// TIA Portal project "traffic_light" (V17)

(* hardware
DEVICE "S7-1200 station_1"  S7-1200 Station
   slot 0: "Rack_0"  S7-1200 Rack  Rack  V1.0
   slot 1: "PLC_1"  CPU 1212C DC/DC/DC  6ES7 212-1AE40-0XB0  V4.1
DEVICE "HMI_1"  TP700 Comfort
   slot 0: "HMI_1"  TP700 Comfort  6AV2 124-0GC01-0AX0  17.0.0.0
   slot 1: "HMI_RT_1"  TP700 Comfort  6AV2 124-0GC01-0AX0  17.0.0.0
   slot 5: "HMI_1.IE_CP_1"  PROFINET Interface  17.0.0.0
      slot 1: "PROFINET Interface_1"  PROFINET Interface
         slot 1: "Port_1"  Port
         slot 2: "Port_2"  Port
   slot 7: "HMI_1.MPI/DP_CP_1"  MPI/DP Interface  17.0.0.0
*)

// ===== PLC "PLC_1"  CPU 1212C DC/DC/DC =====

VAR_GLOBAL   // PLC tag table "Tag table_1"
   "START" AT %M0.0 : Bool;
   "STOP" AT %M0.1 : Bool;
   "STARTED" AT %M0.2 : Bool;
   "STEP1_EAST_GREEN" AT %M0.3 : Bool;
   "STEP1_WEST_RED" AT %M0.4 : Bool;
   "STEP1_NORTH_RED" AT %M0.5 : Bool;
   "STEP1_EAST_YELLOW" AT %M0.6 : Bool;
   "STEP1_FINISHED" AT %M0.7 : Bool;
   "STEP2_WEST_GREEN" AT %M1.0 : Bool;
   "STEP2_EAST_RED" AT %M1.1 : Bool;
   "STEP2_NORTH_RED" AT %M1.2 : Bool;
   "STEP2_WEST_YELLOW" AT %M1.3 : Bool;
   "STEP2_FINISHED" AT %M1.4 : Bool;
   "STEP3_NORTH_GREEN" AT %M1.5 : Bool;
   "STEP3_WEST_RED" AT %M1.6 : Bool;
   "STEP3_EAST_RED" AT %M1.7 : Bool;
   "STEP3_NORTH_YELLOW" AT %M2.0 : Bool;
   "STEP3_FINISHED" AT %M2.1 : Bool;
   "EAST_GREEN" AT %M2.2 : Bool;
   "EAST_YELLOW" AT %M2.3 : Bool;
   "EAST_RED" AT %M2.4 : Bool;
   "NORTH_RED" AT %M2.5 : Bool;
   "NORTH_GREEN" AT %M2.6 : Bool;
   "NORTH_YELLOW" AT %M2.7 : Bool;
   "WEST_RED" AT %M3.0 : Bool;
   "WEST_GREEN" AT %M3.1 : Bool;
   "WEST_YELLOW" AT %M3.2 : Bool;
END_VAR

// folder: System blocks/Program resources

DATA_BLOCK "STEP1"   // DB1
{ S7_Optimized_Access := 'TRUE' }
AUTHOR : Simatic
FAMILY : IEC
NAME : IEC_TMR
VERSION : 1.0
// stored: InstanceOfName IEC_TIMER
"IEC_TIMER"
BEGIN
END_DATA_BLOCK

DATA_BLOCK "COUNTER_STEP"   // DB2
{ S7_Optimized_Access := 'TRUE' }
AUTHOR : Simatic
FAMILY : IEC
NAME : CNTR
VERSION : 1.0
// stored: InstanceOfName IEC_COUNTER
"IEC_COUNTER"
BEGIN
END_DATA_BLOCK

DATA_BLOCK "STEP2"   // DB3
{ S7_Optimized_Access := 'TRUE' }
AUTHOR : Simatic
FAMILY : IEC
NAME : IEC_TMR
VERSION : 1.0
// stored: InstanceOfName IEC_TIMER
"IEC_TIMER"
BEGIN
END_DATA_BLOCK

DATA_BLOCK "STEP3"   // DB4
{ S7_Optimized_Access := 'TRUE' }
AUTHOR : Simatic
FAMILY : IEC
NAME : IEC_TMR
VERSION : 1.0
// stored: InstanceOfName IEC_TIMER
"IEC_TIMER"
BEGIN
END_DATA_BLOCK

// folder: (top level)

ORGANIZATION_BLOCK "Main"   // OB1, LAD, ProgramCycle
TITLE = "Main Program Sweep (Cycle)"
{ S7_Optimized_Access := 'TRUE' }
VERSION : 0.1
   VAR_INPUT
      Initial_Call : Bool;   // Initial call of this OB
      Remanence : Bool;   // =True, if remanent data are available
   END_VAR
   VAR_TEMP   // added for the SCL form of the ladder/FBD networks
      _w1 : Bool;
      _w2 : Bool;
      _w3 : Bool;
   END_VAR
BEGIN

REGION Network 1
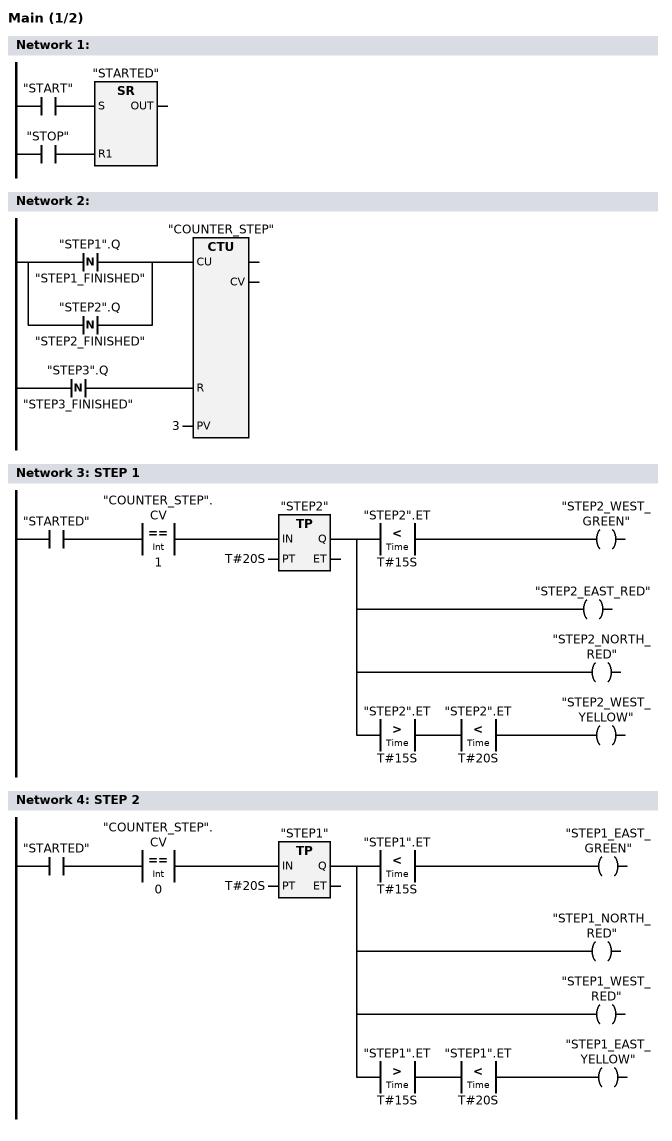
   RUNG wire#powerrail
      Contact( "START" )
      S_SR(operand := "STARTED", r1 := wire#w1)
   END_RUNG
   RUNG wire#powerrail
      Contact( "STOP" )
   END_RUNG wire#w1
   // the same network as SCL:
   IF "START" THEN
       "STARTED" := TRUE;   // SR flip-flop
   END_IF;
   IF "STOP" THEN "STARTED" := FALSE; END_IF;
END_REGION

REGION Network 2
   #_w1 := NOT "STEP1".Q AND "STEP1_FINISHED";   // falling edge of "STEP1".Q
   "STEP1_FINISHED" := "STEP1".Q;
   #_w2 := NOT "STEP2".Q AND "STEP2_FINISHED";   // falling edge of "STEP2".Q
   "STEP2_FINISHED" := "STEP2".Q;
   #_w3 := NOT "STEP3".Q AND "STEP3_FINISHED";   // falling edge of "STEP3".Q
   "STEP3_FINISHED" := "STEP3".Q;
   "COUNTER_STEP".CTU(CU := #_w1 OR #_w2, R := #_w3, PV := 3);
END_REGION

REGION Network 3: STEP 1
   "STEP2".TP(IN := "STARTED" AND ("COUNTER_STEP".CV = 1), PT := T#20S);
   "STEP2_WEST_GREEN" := "STEP2".Q AND ("STEP2".ET < T#15S);
   "STEP2_EAST_RED" := "STEP2".Q;
   "STEP2_NORTH_RED" := "STEP2".Q;
   "STEP2_WEST_YELLOW" := "STEP2".Q AND ("STEP2".ET > T#15S) AND ("STEP2".ET < T#20S);
END_REGION

REGION Network 4: STEP 2
   "STEP1".TP(IN := "STARTED" AND ("COUNTER_STEP".CV = 0), PT := T#20S);
   "STEP1_EAST_GREEN" := "STEP1".Q AND ("STEP1".ET < T#15S);
   "STEP1_NORTH_RED" := "STEP1".Q;
   "STEP1_WEST_RED" := "STEP1".Q;
   "STEP1_EAST_YELLOW" := "STEP1".Q AND ("STEP1".ET > T#15S) AND ("STEP1".ET < T#20S);
END_REGION

REGION Network 5: STEP3
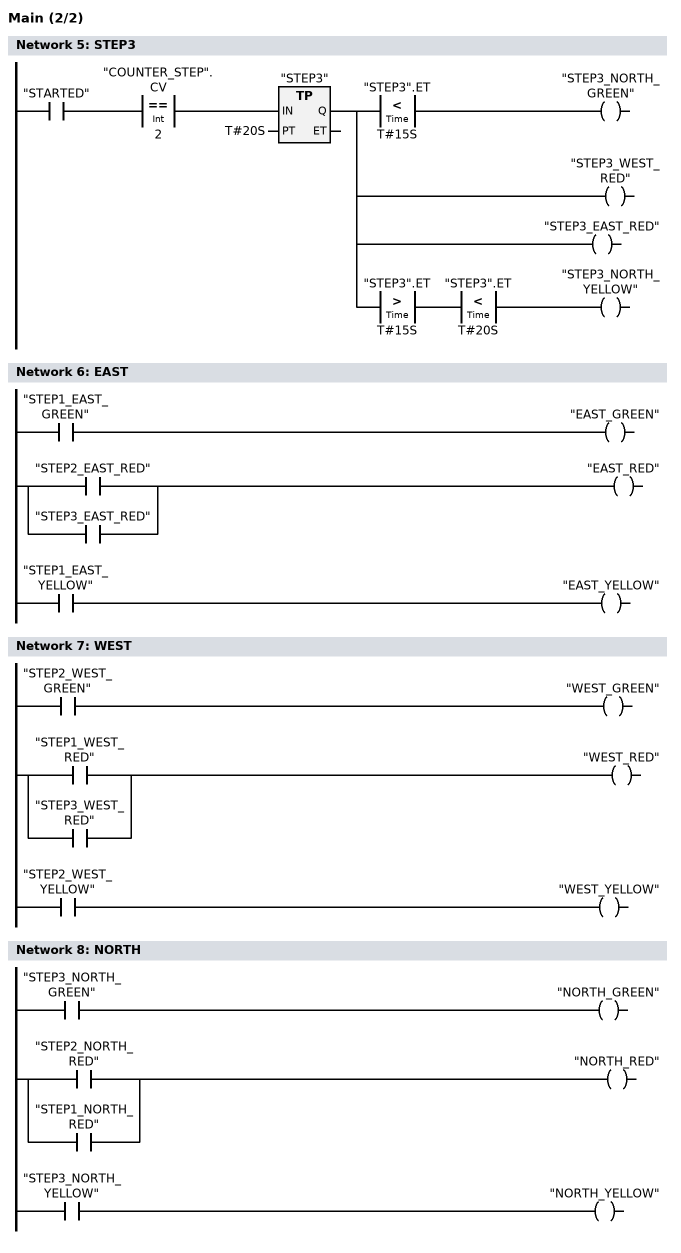
   "STEP3".TP(IN := "STARTED" AND ("COUNTER_STEP".CV = 2), PT := T#20S);
   "STEP3_NORTH_GREEN" := "STEP3".Q AND ("STEP3".ET < T#15S);
   "STEP3_WEST_RED" := "STEP3".Q;
   "STEP3_EAST_RED" := "STEP3".Q;
   "STEP3_NORTH_YELLOW" := "STEP3".Q AND ("STEP3".ET > T#15S) AND ("STEP3".ET < T#20S);
END_REGION

REGION Network 6: EAST
   RUNG wire#powerrail
      Contact( "STEP1_EAST_GREEN" )
      Coil( "EAST_GREEN" )
   END_RUNG
   RUNG wire#powerrail
      Contact( "STEP2_EAST_RED" )
      wire#w1
      Coil( "EAST_RED" )
   END_RUNG
   RUNG wire#powerrail
      Contact( "STEP3_EAST_RED" )
   END_RUNG wire#w1
   RUNG wire#powerrail
      Contact( "STEP1_EAST_YELLOW" )
      Coil( "EAST_YELLOW" )
   END_RUNG
   // the same network as SCL:
   "EAST_GREEN" := "STEP1_EAST_GREEN";
   "EAST_RED" := "STEP2_EAST_RED" OR "STEP3_EAST_RED";
   "EAST_YELLOW" := "STEP1_EAST_YELLOW";
END_REGION

REGION Network 7: WEST
   RUNG wire#powerrail
      Contact( "STEP2_WEST_GREEN" )
      Coil( "WEST_GREEN" )
   END_RUNG
   RUNG wire#powerrail
      Contact( "STEP1_WEST_RED" )
      wire#w1
      Coil( "WEST_RED" )
   END_RUNG
   RUNG wire#powerrail
      Contact( "STEP3_WEST_RED" )
   END_RUNG wire#w1
   RUNG wire#powerrail
      Contact( "STEP2_WEST_YELLOW" )
      Coil( "WEST_YELLOW" )
   END_RUNG
   // the same network as SCL:
   "WEST_GREEN" := "STEP2_WEST_GREEN";
   "WEST_RED" := "STEP1_WEST_RED" OR "STEP3_WEST_RED";
   "WEST_YELLOW" := "STEP2_WEST_YELLOW";
END_REGION

REGION Network 8: NORTH
   RUNG wire#powerrail
      Contact( "STEP3_NORTH_GREEN" )
      Coil( "NORTH_GREEN" )
   END_RUNG
   RUNG wire#powerrail
      Contact( "STEP2_NORTH_RED" )
      wire#w1
      Coil( "NORTH_RED" )
   END_RUNG
   RUNG wire#powerrail
      Contact( "STEP1_NORTH_RED" )
   END_RUNG wire#w1
   RUNG wire#powerrail
      Contact( "STEP3_NORTH_YELLOW" )
      Coil( "NORTH_YELLOW" )
   END_RUNG
   // the same network as SCL:
   "NORTH_GREEN" := "STEP3_NORTH_GREEN";
   "NORTH_RED" := "STEP2_NORTH_RED" OR "STEP1_NORTH_RED";
   "NORTH_YELLOW" := "STEP3_NORTH_YELLOW";
END_REGION
END_ORGANIZATION_BLOCK

(* ===== HMI "HMI_RT_1" =====
system functions are stored by id; their names below are inferred from use
connection "HMI_Connection_1": ETHERNET, S7_1200_OMS

HMI tags "Default tag table"
   "WEST_GREEN" : Bool = PLC WEST_GREEN AT %M3.1, 1 s
   "WEST_YELLOW" : Bool = PLC WEST_YELLOW AT %M3.2, 1 s
   "WEST_RED" : Bool = PLC WEST_RED AT %M3.0, 1 s
   "STEP3_NORTH_GREEN" : Bool = PLC STEP3_NORTH_GREEN AT %M1.5, 1 s
   "NORTH_GREEN" : Bool = PLC NORTH_GREEN AT %M2.6, 1 s
   "NORTH_YELLOW" : Bool = PLC NORTH_YELLOW AT %M2.7, 1 s
   "NORTH_RED" : Bool = PLC NORTH_RED AT %M2.5, 1 s
   "EAST_GREEN" : Bool = PLC EAST_GREEN AT %M2.2, 1 s
   "EAST_YELLOW" : Bool = PLC EAST_YELLOW AT %M2.3, 1 s
   "EAST_RED" : Bool = PLC EAST_RED AT %M2.4, 1 s
   "START" : Bool = PLC START AT %M0.0, 1 s
   "STOP" : Bool = PLC STOP AT %M0.1, 1 s

screen "Screen_1" 800x480
   GraphicView "Graphic view_1" at 0,0 size 678x368; Picture "3-way-traffic-light-control-ladder-logic-removebg-preview"
   Circle "Circle_1" at 329,228 size 19x19
      Appearance <- "NORTH_GREEN"
   Circle "Circle_2" at 352,228 size 19x19
      Appearance <- "NORTH_YELLOW"
   Circle "Circle_3" at 374,228 size 19x19
      Appearance <- "NORTH_RED"
   Circle "Circle_4" at 278,236 size 19x19
      Appearance <- "WEST_GREEN"
   Circle "Circle_5" at 278,283 size 19x19
      Appearance <- "WEST_RED"
   Circle "Circle_6" at 278,259 size 19x19
      Appearance <- "WEST_YELLOW"
   Circle "Circle_7" at 389,270 size 19x19
      Appearance <- "EAST_GREEN"
   Circle "Circle_8" at 389,294 size 19x19
      Appearance <- "EAST_YELLOW"
   Circle "Circle_9" at 389,318 size 19x19
      Appearance <- "EAST_RED"
   Button "Button_1" at 75,399 size 96x32; TextOff 'START'
      on Release: ResetBit("START")
      on Press: SetBit("START")
   Button "Button_2" at 231,399 size 96x32; TextOff 'STOP'
      on Press: SetBit("STOP")
      on Release: ResetBit("STOP")
   GraphicView "Graphic view_2" at 470,26 size 245x182; Picture "Screenshot 2025-08-15 150041"
*)